// TIA Portal V20 export
// export: Created 2025-12-01T14:56:18.1245367Z, ExportSetting None, DisplayName Totally Integrated Automation Portal, DisplayVersion V20 Update 3, DisplayName TIA Portal Openness, DisplayVersion V20 Update 3, DisplayName TIA Portal Version Control Interface, DisplayVersion V20 Update 3, DisplayName STEP 7 Professional, DisplayVersion V20 Update 3, DisplayName STEP 7 Safety, DisplayVersion V20 Update 2, DisplayName WinCC Basic/Comfort/Advanced, DisplayVersion V20 Update 3, DisplayName WinCC Professional, DisplayVersion V20 Update 3, DisplayName WinCC Unified, DisplayVersion V20 Update 3
TYPE "Danfoss_STW_PN"
   STRUCT
      Speed_Ok : Bool;
      Bus_Control : Bool;
      Frecuency_Limit_Ok : Bool;
      In_Operation : Bool;
      N_Drive_Ok : Bool;   // Si esta False siginifica que esta Ok
      Voltage_Excedeed : Bool;
      Toque_Exceeded : Bool;
      Timer_Exceeded : Bool;
      Control_Ready : Bool;
      Drive_Ready : Bool;
      Enable : Bool;
      Trip : Bool;
      ON2 : Bool;
      ON3 : Bool;
      Start_not_Possible : Bool;
      Warning : Bool;
   END_STRUCT;
END_TYPE
